FUNCTION_BLOCK FeedInfluentLogic (* CAT Function Block Type *)
  (* Standard: 61499-2 *)
  (* Version 0.0, 6/13/2026, Schneider Electric, template *)
  PACKAGE SE.Nereda;
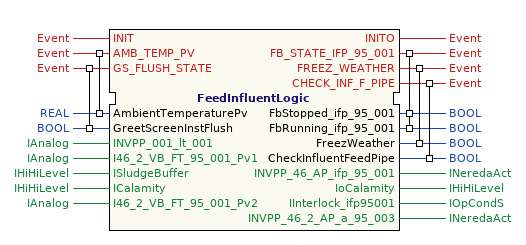
  EVENT_INPUT
    INIT;
    AMB_TEMP_PV WITH AmbientTemperaturePv;
    GS_FLUSH_STATE WITH GreetScreenInstFlush;
  END_EVENT
  EVENT_OUTPUT
    INITO;
    FB_STATE_IFP_95_001 WITH FbStopped_ifp_95_001, FbRunning_ifp_95_001;
    FREEZ_WEATHER WITH FreezWeather; (* Input changed *)
    CHECK_INF_F_PIPE WITH CheckInfluentFeedPipe;
  END_EVENT
  VAR_INPUT
    AmbientTemperaturePv : REAL;
    GreetScreenInstFlush : BOOL;
  END_VAR
  VAR_OUTPUT
    FbStopped_ifp_95_001 : BOOL;
    FbRunning_ifp_95_001 : BOOL;
    FreezWeather : BOOL; (* Output value *)
    CheckInfluentFeedPipe : BOOL;
  END_VAR
  SOCKETS
    INVPP_001_lt_001 : IAnalog;
    I46_2_VB_FT_95_001_Pv1 : IAnalog;
    ISludgeBuffer : IHiHiLevel;
    ICalamity : IHiHiLevel;
  END_SOCKETS
  SOCKETS
    I46_2_VB_FT_95_001_Pv2 : IAnalog; (* Process value (range considered) interface adapter *)
  END_SOCKETS
  PLUGS
    INVPP_46_AP_ifp_95_001 : INeredaAct;
    IoCalamity : IHiHiLevel;
  END_PLUGS
  PLUGS
    IInterlock_ifp95001 : IOpCondS; (* Condition summary chain output to downstream block *)
    INVPP_46_2_AP_a_95_003 : INeredaAct;
  END_PLUGS
  (* 01 - FUNCTIONNAL INPUT INTERFACE *)
  (* 00 - INITIALIZATION *)
  (* 05 - LOGIC *)
  (* 06 - HMI INTERFACE *)
  (* 03 - FIELD INTERFACE *)
  (* Feed Influent Logic *)
  (* 02 - FUNCTIONNAL OUTPUT INTERFACE *)
  (* Interlock *)
  FBS
    IThis : FeedInfluentLogic_HMI(QI := TRUE);
    FeedInfluentLogic : FeedInfluentBasic;
    _46_2_VB_FT_95_001_Status : decodeStatus; {SET_ATTRIBUTE(Configuration.Component.HideUnusedPorts, )}
    CmdPumpSmooth : boolValueChanged;
    FreezRunOperation : E_DELAY_V_D;
    FreezStopOperation : E_DELAY_V_D;
    FreezWeatherSp : COMPARE_1329C2AB45109BAAB; {SET_ATTRIBUTE(Configuration.GenericFBType.InterfaceParams, Runtime.Standard#CNT:=2;IN${CNT$}:REAL)} {SET_ATTRIBUTE(Configuration.Component.HideUnusedPorts, )}
    FreezWeatherSmooth : boolValueChanged;
    PID : PID; {SET_ATTRIBUTE(Configuration.Component.HideUnusedPorts, )}
    FeedFlowSp : FeedPumpFlowSp;
    LowLowFlow_ifp95001 : ilckCondItem(CondCause := Active1);
    LowLowFlowAlarm : AND_88A3DD8EC65DD11C; {SET_ATTRIBUTE(Configuration.GenericFBType.InterfaceParams, Runtime.Standard#CNT:=2;OUT:BOOL)}
    INVPP_001_lt_001_Status : decodeStatus; {SET_ATTRIBUTE(Configuration.Component.HideUnusedPorts, )}
    HighHighLevel_SB : ilckCondItem(CondCause := Active1);
    HighHighLevel_Calamity : ilckCondItem(CondCause := Active1);
    LevelSwitch_Calamity : ilckCondItem(CondCause := Active1);
    RESET_BTNs : RESET_BTNs;
    LoLoFlowAlarmManager : DelayedActive(pin_4E076A4928A0DFEF := TRUE);
    PIDISc : PID_Manager;
    CmdPump : BOOL2INT;
    ValveControl : OpeningValveDurLogic;
    SpeedSp : SpeedSpFlowSensorFail;
    AutoReset : AutoResetCdt;
    Reset : OR_88A3DD8EC65DD11C; {SET_ATTRIBUTE(Configuration.GenericFBType.InterfaceParams, Runtime.Standard#CNT:=2;OUT:BOOL)}
    StartLevelSp : COMPARE_1329C2AB45109BAAB; {SET_ATTRIBUTE(Configuration.GenericFBType.InterfaceParams, Runtime.Standard#CNT:=2;IN${CNT$}:REAL)}
    Wait : E_DELAY(DT := T#500ms);
  END_FBS
  EVENT_CONNECTIONS
    FreezWeatherSp.CNF TO FreezWeatherSmooth.REQ;
    AMB_TEMP_PV TO FreezWeatherSp.REQ;
    LowLowFlowAlarm.CNF TO LowLowFlow_ifp95001.REQ;
    I46_2_VB_FT_95_001_Pv1.REQ_STATUS TO _46_2_VB_FT_95_001_Status.REQ;
    _46_2_VB_FT_95_001_Status.CNF TO LowLowFlowAlarm.REQ;
    INVPP_001_lt_001.REQ_STATUS TO INVPP_001_lt_001_Status.REQ;
    FreezWeatherSmooth.CHD TO FREEZ_WEATHER;
    INVPP_001_lt_001_Status.CNF TO FeedInfluentLogic.1A10D9AD62D4B5BA;
    GS_FLUSH_STATE TO FeedInfluentLogic.3BB3C8F4542D663C;
    ISludgeBuffer.15126F43E529BB4F TO HighHighLevel_SB.REQ;
    ICalamity.15126F43E529BB4F TO IoCalamity.15126F43E529BB4F;
    ICalamity.15126F43E529BB4F TO LevelSwitch_Calamity.REQ;
    ICalamity.15126F43E529BB4F TO HighHighLevel_Calamity.REQ;
    INVPP_46_AP_ifp_95_001.9CD053F8408797ED TO FB_STATE_IFP_95_001;
    CmdPump.6FC99A5BD1C38561 TO INVPP_46_AP_ifp_95_001.0F1CDF9A9B4A227A;
    SpeedSp.1FEAADE7145F64BE TO INVPP_46_AP_ifp_95_001.1E00729184986247;
    INVPP_46_AP_ifp_95_001.9CD053F8408797ED TO FeedInfluentLogic.FA8D01F8193412B5;
    INVPP_46_AP_ifp_95_001.9CD053F8408797ED TO Reset.REQ;
    INVPP_46_AP_ifp_95_001.CC753684FA882790 TO FeedInfluentLogic.BA18149E37AD28B3;
    FreezRunOperation.INITO TO FreezStopOperation.INIT;
    FreezStopOperation.INITO TO PIDISc.INIT;
    PIDISc.CE80458C9D5EF15A TO ValveControl.B0D405FAB24B1E1C;
    FeedInfluentLogic.A886049003AB7BF0 TO CmdPumpSmooth.REQ;
    CmdPumpSmooth.CHD TO CmdPump.DD5870AA881150BB;
    FeedInfluentLogic.A36A5BFEC9789D92 TO FreezRunOperation.START;
    FeedInfluentLogic.DAFC9A25279F77FA TO FreezRunOperation.STOP;
    FeedInfluentLogic.FE42F39B20F05254 TO FreezStopOperation.START;
    FeedInfluentLogic.4542C2B348B73018 TO FreezStopOperation.STOP;
    FreezRunOperation.1457E63E0C241C83 TO FeedInfluentLogic.A841DEC9A7185651;
    FreezStopOperation.1457E63E0C241C83 TO FeedInfluentLogic.BF17A06E73262AF1;
    FreezWeatherSmooth.CHD TO FeedInfluentLogic.0C4F94A66BD0D588;
    INVPP_001_lt_001.REQ TO FeedFlowSp.REQ_LEVEL;
    FeedFlowSp.CNF_FLOW_SP TO PIDISc.REQ;
    CmdPump.6FC99A5BD1C38561 TO PIDISc.REQ;
    LoLoFlowAlarmManager.DDA64CDC00519DA4 TO LowLowFlowAlarm.REQ;
    INVPP_001_lt_001.REQ TO FeedInfluentLogic.087CD876DCD6EE87;
    INIT TO IThis.DA969393F6D27920;
    FeedInfluentLogic.773D179CB48D8BCF TO IThis.ACDDFE951F9AC365;
    IThis.CF4D33127CB86F75 TO IThis.6FEE224494FEC59A;
    ISludgeBuffer.15126F43E529BB4F TO IThis.0B15839312D7291F;
    ICalamity.15126F43E529BB4F TO IThis.0B15839312D7291F;
    PIDISc.CE80458C9D5EF15A TO IThis.0B15839312D7291F;
    FreezWeatherSmooth.CHD TO IThis.26057A70B314F6D6;
    RESET_BTNs.920962203CA54948 TO IThis.2C41FD5D4355E4C3;
    PIDISc.CE80458C9D5EF15A TO IThis.3D88186A4172EAF0;
    IThis.A8EF0BC2917800E0 TO FreezRunOperation.INIT;
    IThis.3F66EB998062A9C8 TO FreezRunOperation.8C325F07198FCB13;
    IThis.3F66EB998062A9C8 TO FreezStopOperation.8C325F07198FCB13;
    IThis.72B00C04BD02DD2F TO FreezWeatherSp.REQ;
    IThis.FBAAF03BEE48839D TO FeedInfluentLogic.D9F01C23F33FA44E;
    IThis.FBAAF03BEE48839D TO RESET_BTNs.AB695E9A35A20E19;
    IThis.CF4D33127CB86F75 TO FeedFlowSp.REQ_LEVEL;
    IThis.CF4D33127CB86F75 TO FeedInfluentLogic.087CD876DCD6EE87;
    IThis.3306829F90F658EB TO Reset.REQ;
    IThis.3306829F90F658EB TO RESET_BTNs.AB695E9A35A20E19;
    ValveControl.599C3061E75F42AF TO AutoReset.59F74AF1EC48CDE2;
    INVPP_46_AP_ifp_95_001.9CD053F8408797ED TO ValveControl.D723ED8511816BBA;
    PID.CNF TO SpeedSp.B5D6B08FA2666F02;
    _46_2_VB_FT_95_001_Status.CNF TO SpeedSp.B5D6B08FA2666F02;
    I46_2_VB_FT_95_001_Pv1.REQ TO SpeedSp.B5D6B08FA2666F02;
    FeedFlowSp.CNF_FLOW_SP TO SpeedSp.B5D6B08FA2666F02;
    AutoReset.64AA955A8D38780A TO INITO;
    LowLowFlowAlarm.CNF TO AutoReset.9806DB285215C1DB;
    AutoReset.F95261E270E5ADCA TO Reset.REQ;
    Reset.CNF TO LoLoFlowAlarmManager.C451626F7187F42D;
    AutoReset.9201C3DE5912C4B7 TO CHECK_INF_F_PIPE;
    StartLevelSp.CNF TO AutoReset.9B7806BCABA1FC1F;
    IThis.CF4D33127CB86F75 TO StartLevelSp.REQ;
    INVPP_001_lt_001.REQ TO StartLevelSp.REQ;
    IThis.3306829F90F658EB TO AutoReset.455A9133E8D25793;
    FeedInfluentLogic.462EBC5E04F2E8AC TO Wait.START;
    Wait.EO TO FeedInfluentLogic.A6EDF9258529D74A;
  END_CONNECTIONS
  DATA_CONNECTIONS
    FreezWeatherSp.LE TO FreezWeatherSmooth.Input;
    AmbientTemperaturePv TO FreezWeatherSp.IN1;
    I46_2_VB_FT_95_001_Pv1.Status TO _46_2_VB_FT_95_001_Status.Status;
    _46_2_VB_FT_95_001_Status.LoLoAlarm TO LowLowFlowAlarm.IN2;
    INVPP_001_lt_001.Status TO INVPP_001_lt_001_Status.Status;
    FreezWeatherSmooth.Output TO FreezWeather;
    INVPP_001_lt_001_Status.HiAlarm TO FeedInfluentLogic.CCE17708114D7274;
    GreetScreenInstFlush TO FeedInfluentLogic.5B7FAD7223786DCB;
    ICalamity.C818324478A2F205 TO IoCalamity.C818324478A2F205;
    ICalamity.96B50ADF37756FFC TO IoCalamity.96B50ADF37756FFC;
    INVPP_46_AP_ifp_95_001.D83B5BDEFA4D797C TO FbStopped_ifp_95_001;
    INVPP_46_AP_ifp_95_001.B762734C094A7162 TO FbRunning_ifp_95_001;
    CmdPump.A6DEF5F9C27C1848 TO INVPP_46_AP_ifp_95_001.710D7FC54EE3F35A;
    SpeedSp.87931CA83794BFFD TO INVPP_46_AP_ifp_95_001.1BC103921BBFDA0B;
    INVPP_46_AP_ifp_95_001.D83B5BDEFA4D797C TO FeedInfluentLogic.F46B1546E818D164;
    INVPP_46_AP_ifp_95_001.B762734C094A7162 TO FeedInfluentLogic.A435A18234D11579;
    INVPP_46_AP_ifp_95_001.B762734C094A7162 TO LoLoFlowAlarmManager.19546B227DE05AED;
    INVPP_46_AP_ifp_95_001.8A8A07EFCDA1443C TO FeedInfluentLogic.D3CC68030E716A58;
    CmdPumpSmooth.Output TO CmdPump.4573FC8F228EB71D;
    FeedInfluentLogic.6FD1A8945A6CB7E1 TO CmdPumpSmooth.Input;
    CmdPumpSmooth.Output TO PIDISc.RunPID;
    FreezRunOperation.716D3F3042596C89 TO FeedInfluentLogic.9E484CF026FEE50F;
    FreezStopOperation.716D3F3042596C89 TO FeedInfluentLogic.4DA8AA650AC4FC55;
    FreezWeatherSmooth.Output TO FeedInfluentLogic.D6D1DFF1CBB2AE71;
    INVPP_001_lt_001.Value TO FeedFlowSp.InfluentLevel;
    FeedFlowSp.FlowSp TO PIDISc.Setpoint;
    LoLoFlowAlarmManager.614F3125208254F6 TO LowLowFlowAlarm.IN1;
    INVPP_001_lt_001.Value TO FeedInfluentLogic.4E1A1BF0C390C99A;
    FeedInfluentLogic.4CDD3E3012708AFD TO IThis.B8642C11FD7EB72C;
    IThis.BDE03EDBA9A0A397 TO IThis.9F798F3C0A181FC5;
    IThis.37384081B1607599 TO IThis.987670AFD4AF32B0;
    IThis.85BDF3D9DCBC4E5E TO IThis.9960B57FC3A75D13;
    ISludgeBuffer.C818324478A2F205 TO IThis.259A079AF3442847;
    ICalamity.C818324478A2F205 TO IThis.C4E8CF1A9E1E6A19;
    ICalamity.96B50ADF37756FFC TO IThis.F8F483ACE30DC46D;
    FreezWeatherSmooth.Output TO IThis.91B0609076B410EA;
    IThis.F7CC81D7079C77C4 TO FreezRunOperation.DT1;
    IThis.C81E5CA34DAFD21D TO FreezStopOperation.DT1;
    IThis.854468E32F5202B4 TO FreezWeatherSp.IN2;
    IThis.5677B89D58E0B562 TO FeedInfluentLogic.A37751783FF88338;
    IThis.5677B89D58E0B562 TO RESET_BTNs.26767209E3135B52;
    IThis.BDE03EDBA9A0A397 TO FeedFlowSp.StartLevelSp;
    IThis.BDE03EDBA9A0A397 TO FeedInfluentLogic.C449D5A81D824C6A;
    IThis.37384081B1607599 TO FeedFlowSp.StopLevelSp;
    IThis.37384081B1607599 TO FeedInfluentLogic.4B0410BD252B6697;
    IThis.85BDF3D9DCBC4E5E TO FeedFlowSp.BreakPoint;
    IThis.67FBC335D0B2273D TO FeedFlowSp.MaxFlowSP;
    IThis.40A923BA8E60A623 TO LoLoFlowAlarmManager.1CE054BDD0AD4DEB;
    IThis.FA45CE8B7738EAEF TO Reset.IN1;
    IThis.FA45CE8B7738EAEF TO RESET_BTNs.479D4538AEFD6EE1;
    INVPP_46_AP_ifp_95_001.B762734C094A7162 TO ValveControl.859CB6DCE329D25D;
    INVPP_46_AP_ifp_95_001.D83B5BDEFA4D797C TO ValveControl.985B4AC3F5EAC315;
    _46_2_VB_FT_95_001_Status.FailAlarm TO SpeedSp.1C28FEF37A13F67F;
    I46_2_VB_FT_95_001_Pv1.ValueMax TO SpeedSp.75C86D8B7647050C;
    I46_2_VB_FT_95_001_Pv1.ValueMin TO SpeedSp.B08827D02DBBFA97;
    FeedFlowSp.FlowSp TO SpeedSp.3BE251DFC2E7905D;
    PID.Out TO SpeedSp.4727B0C2E5DD09FB;
    LowLowFlowAlarm.OUT TO AutoReset.BB8588719CFB4FFD;
    AutoReset.33F44F8BA0B61F91 TO Reset.IN2;
    Reset.OUT TO LoLoFlowAlarmManager.45767490F5BA3A44;
    AutoReset.4E94A160674F4D2C TO CheckInfluentFeedPipe;
    StartLevelSp.LE TO AutoReset.E7812FAD3E29EA1C;
    INVPP_001_lt_001.Value TO StartLevelSp.IN1;
    IThis.BDE03EDBA9A0A397 TO StartLevelSp.IN2;
    IThis.FA45CE8B7738EAEF TO AutoReset.75B143383ED74CE4;
  END_CONNECTIONS
  ADAPTER_CONNECTIONS
    I46_2_VB_FT_95_001_Pv2 TO PID.IPv;
    LowLowFlow_ifp95001.ICondChainOut TO IInterlock_ifp95001;
    HighHighLevel_Calamity.ICondChainOut TO HighHighLevel_SB.ICondChainIn;
    LevelSwitch_Calamity.ICondChainOut TO HighHighLevel_Calamity.ICondChainIn;
    HighHighLevel_SB.ICondChainOut TO LowLowFlow_ifp95001.ICondChainIn;
    PIDISc.FACD1DD4E791A86A TO PID.ISc;
    ValveControl.F83096AD3BF61126 TO INVPP_46_2_AP_a_95_003;
  END_CONNECTIONS
END_FUNCTION_BLOCK
